{attribute addProperty BoxType "EP9224-0037-0017"}
{attribute addProperty Id "DPO_Inputs_ChannelAT %I*ARRAY[0..3] OF DPO_Inputs_Channel_AD3CD21C192240DPO_Inputs_DeviceAT %I*DPO_Inputs_Device_C2311DBA96120DPO_Outputs_ChannelAT %Q*ARRAY[0..3] OF DPO_Outputs_Channel_5760563F128160DPO_Outputs_DeviceAT %Q*DPO_Outputs_Device_6EB864581620WcStateAT %I*WcState_F855686C1620InfoDataAT %I*InfoData_0BDED7BF144180"}
{attribute addProperty CRC "875509549"}
{attribute addProperty SizeInBites "592"}
{attribute addProperty SizeInBytes "74"}
TYPE EP9224_D011B61C :
STRUCT
	{attribute addProperty Name "DPO_Inputs_Channel"}
	DPO_Inputs_Channel : ARRAY[0..3] OF DPO_Inputs_Channel_AD3CD21C;
	{attribute addProperty Name "DPO_Inputs_Device"}
	DPO_Inputs_Device : DPO_Inputs_Device_C2311DBA;
	{attribute addProperty Name "DPO_Outputs_Channel"}
	DPO_Outputs_Channel : ARRAY[0..3] OF DPO_Outputs_Channel_5760563F;
	{attribute addProperty Name "DPO_Outputs_Device"}
	DPO_Outputs_Device : DPO_Outputs_Device_6EB86458;
	{attribute addProperty Name "WcState"}
	WcState : WcState_F855686C;
	{attribute addProperty Name "InfoData"}
	InfoData : InfoData_0BDED7BF;
END_STRUCT
END_TYPE

(* stored: Version 1.2.0.0, ProductVersion 3.1.4024.9
   DUT EP9224_D011B61C: Id {b8beca15-68b9-481e-81a5-b51062e25b93} *)
